// TIA Portal V17 export
// export: Created 2024-09-02T12:49:53.8959663Z, ExportSetting WithDefaults, DisplayName Totally Integrated Automation Portal, DisplayVersion V17, DisplayName TIA Portal Openness, DisplayVersion V17, DisplayName TIA Portal Version Control Interface, DisplayVersion V17, DisplayName STEP 7 Professional, DisplayVersion V17, DisplayName STEP 7 Safety, DisplayVersion V17, DisplayName WinCC Professional, DisplayVersion V17
FUNCTION "AnwFC_Safety_Info" : Void   // FC7002, LAD
TITLE = Safty Info / Safety Info
{ S7_Optimized_Access := 'TRUE' }
AUTHOR : OlegFuehrus
FAMILY : Safe
NAME : Safe
VERSION : 0.1
// stored: AutoNumber true, IsIECCheckEnabled false, SetENOAutomatically false, UDAEnableTagReadback false
   VAR_TEMP
      t_VKE0 : Bool;
      t_VKE1 : Bool;
      t_Signatur_ASCII : Array[1..8] of Char;
      t_RetVal : Word;
   END_VAR
BEGIN

REGION Network 1: INIT
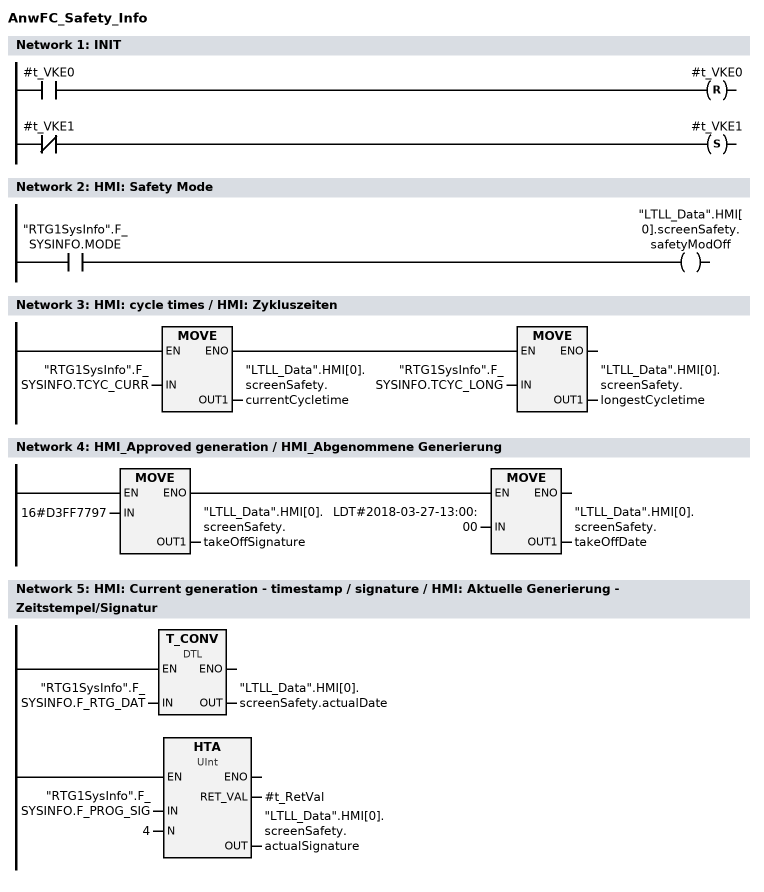
   RUNG wire#powerrail
      Contact( #t_VKE0 )
      R_Coil( #t_VKE0 )
   END_RUNG
   RUNG wire#powerrail
      I_Contact( #t_VKE1 )
      S_Coil( #t_VKE1 )
   END_RUNG
   // the same network as SCL:
   IF #t_VKE0 THEN #t_VKE0 := FALSE; END_IF;
   IF NOT #t_VKE1 THEN #t_VKE1 := TRUE; END_IF;
END_REGION

REGION Network 2: HMI: Safety Mode
   RUNG wire#powerrail
      Contact( "RTG1SysInfo".F_SYSINFO.MODE )
      Coil( "LTLL_Data".HMI[0].screenSafety.safetyModOff )
   END_RUNG
   // the same network as SCL:
   "LTLL_Data".HMI[0].screenSafety.safetyModOff := "RTG1SysInfo".F_SYSINFO.MODE;
END_REGION

REGION Network 3: HMI: cycle times / HMI: Zykluszeiten
   RUNG wire#powerrail
      Move(in := "RTG1SysInfo".F_SYSINFO.TCYC_CURR, out1 => "LTLL_Data".HMI[0].screenSafety.currentCycletime)
      Move(in := "RTG1SysInfo".F_SYSINFO.TCYC_LONG, out1 => "LTLL_Data".HMI[0].screenSafety.longestCycletime)
   END_RUNG
   // the same network as SCL:
   "LTLL_Data".HMI[0].screenSafety.currentCycletime := "RTG1SysInfo".F_SYSINFO.TCYC_CURR;
   "LTLL_Data".HMI[0].screenSafety.longestCycletime := "RTG1SysInfo".F_SYSINFO.TCYC_LONG;
END_REGION

REGION Network 4: HMI_Approved generation / HMI_Abgenommene Generierung
   RUNG wire#powerrail
      Move(in := 16#D3FF7797, out1 => "LTLL_Data".HMI[0].screenSafety.takeOffSignature)
      Move(in := LDT#2018-03-27-13:00:00, out1 => "LTLL_Data".HMI[0].screenSafety.takeOffDate)
   END_RUNG
   // the same network as SCL:
   "LTLL_Data".HMI[0].screenSafety.takeOffSignature := 16#D3FF7797;
   "LTLL_Data".HMI[0].screenSafety.takeOffDate := LDT#2018-03-27-13:00:00;
END_REGION

REGION Network 5: HMI: Current generation - timestamp / signature / HMI: Aktuelle Generierung - Zeitstempel/Signatur
   RUNG wire#powerrail
      { S7_Templates := "[src_type := DTL, dest_type := LDT]" } T_CONV(IN := "RTG1SysInfo".F_SYSINFO.F_RTG_DAT, OUT => "LTLL_Data".HMI[0].screenSafety.actualDate)
   END_RUNG
   RUNG wire#powerrail
      { S7_Templates := "[card := 1, n_type := UInt, in_out_type := Variant]" } HTA(IN := "RTG1SysInfo".F_SYSINFO.F_PROG_SIG, N := 4, RET_VAL => #t_RetVal, OUT => "LTLL_Data".HMI[0].screenSafety.actualSignature)
   END_RUNG
   // the same network as SCL:
   T_CONV(IN := "RTG1SysInfo".F_SYSINFO.F_RTG_DAT, OUT => "LTLL_Data".HMI[0].screenSafety.actualDate);
   #t_RetVal := HTA(IN := "RTG1SysInfo".F_SYSINFO.F_PROG_SIG,
                    N := 4,
                    OUT => "LTLL_Data".HMI[0].screenSafety.actualSignature);
END_REGION
END_FUNCTION
